RoboDK station: PluginAttachObject.rdk

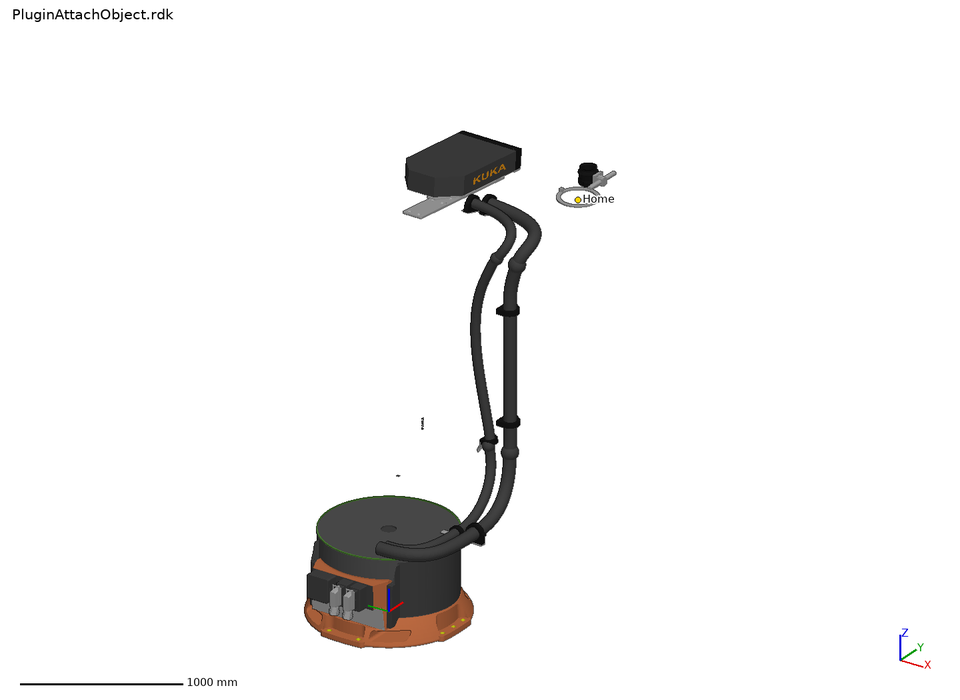
[picture v0: the station drawn from its stored meshes, robots at their saved joint values, targets as dots, program paths as lines]
Station PluginAttachObject (saved by RoboDK 5.3.3). Poses are relative to the parent item; angles as X-Y-Z fixed-axis rotations.
  - frame KUKA KR 480 R3330 MT-F K Base at (0, 0, 0) mm, rotated rx 0 ry 0 rz 90 deg
    - robot KUKA KR 480 R3330 MT-F K: 6 axes, payload 480 kg, reach 3326 mm, repeatability 0.08 mm, weight 2475 kg
        joint limits [-185, -130, -100, -350, -120, -350] to [185, 20, 144, 350, 120, 350]; home [0, -90, 90, 0, 0, 0]; saved at [0, -90, 90, 0, 90, 0]
    - object J1 Cables at (0, 0, 0) mm, size 1030.8 x 764.9 x 504.6 mm
    - object J2 Cables at (0, 0, 0) mm, size 134.9 x 397.5 x 1398 mm
    - object J4 Cables and supply system at (0, 0, 0) mm, size 1113.1 x 1047.4 x 407.8 mm
    - object J6 Cable holder at (-265, 0, 4315) mm, rotated rx 0 ry 90 rz 0 deg, size 117 x 300.5 x 521.3 mm
    - target Home (joint target) at (2025, 0, 2000) mm, rotated rx 180 ry 0 rz -180 deg; joints [0, -90, 90, 0, 90, 0] of KUKA KR 480 R3330 MT-F K
  - Python program AutoAttach (listed below)
  - Python program AutoDetach (listed below)

--- Python program AutoAttach ---
from robolink import *  # RoboDK API
from robodk import *  # Robot toolbox

RDK = Robolink()

robot = RDK.ItemUserPick("Select robot", ITEM_TYPE_ROBOT)
objects = RDK.ItemList(ITEM_TYPE_OBJECT, list_names=True)

# Expected format: "Attach", "Joint|Robot|Object|". Attaches Object to Robot at Joint
#                  "Detach", "Object". Detach Object from any Robot
#                  "Detach", "Robot". Detach all Objects from Robot

for obj in objects:

    joint = int(obj[1])
    value = "%i|%s|%s" % (joint, robot.Name(), obj)
    result = RDK.PluginCommand("Plugin Attach Object", "Attach", value)
    RDK.ShowMessage("Attach " + value + " -> " + result, False)

--- Python program AutoDetach ---
from robolink import *  # RoboDK API
from robodk import *  # Robot toolbox

RDK = Robolink()

robot = RDK.ItemUserPick("Select robot", ITEM_TYPE_ROBOT)

# Expected format: "Attach", "Joint|Robot|Object|". Attaches Object to Robot at Joint
#                  "Detach", "Object". Detach Object from any Robot
#                  "Detach", "Robot". Detach all Objects from Robot

value = robot.Name()
result = RDK.PluginCommand("Plugin Attach Object", "Detach", value)
RDK.ShowMessage("Detach " + value + " -> " + result, False)
